# B&R Automation Studio project BaseLD
Automation Studio 4.7.2.98

## Configuration Config1

CPU X20CP1586, AutomationRuntime C4.72, Build 4.1.2, Vc V4.72.0

### IoMap.iom - X20CP1586/IoMap.iom
```iecst
VAR_CONFIG
	::Program1:LEDon AT %QX."X20DOF322".DigitalOutput01;
END_VAR
```

## Logical view

### Program Logical/Program1

#### Cyclic.ld
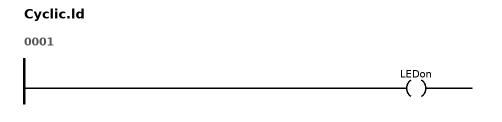
Ladder, written as Structured Text:
```iecst
PROGRAM _CYCLIC
(* Network 1 *)
LEDon := TRUE;
END_PROGRAM
```
